// TIA Portal V18 export
TYPE "PLCtoMES_SubCheckIn_ext"
// stored: IsFailsafeCompliant false
   STRUCT
      Load_SubPart1ChickInReq : Bool;   // 子零件1查询事件触发位
      Load_SubPart2ChickInReq : Bool;   // 子零件2查询事件触发位
      Load_SubPart3ChickInReq : Bool;   // 子零件3查询事件触发位
      Load_SubPart4ChickInReq : Bool;   // 子零件4查询事件触发位
      Load_SubPart5ChickInReq : Bool;   // 子零件5查询事件触发位
      Load_SubPart6ChickInReq : Bool;   // 子零件6查询事件触发位
      Load_SubPart7ChickInReq : Bool;   // 子零件7查询事件触发位
      Load_SubPart8ChickInReq : Bool;   // 子零件8查询事件触发位
   END_STRUCT;
END_TYPE
